FUNCTION_BLOCK FB_MatrixMultiplication
VAR_INPUT
	A : Matrix;
	B : Matrix;
END_VAR
VAR_OUTPUT
	out : Matrix;
END_VAR
VAR
	i : INT;
	j : INT;
	k : INT;
END_VAR

FOR i := 0 TO A.nRows-1 DO
    FOR j := 0 TO B.nCols-1 DO
        out.data[i, j] := 0; 
        FOR k := 0 TO B.nRows-1 DO
            out.data[i, j] := out.data[i, j] + A.data[i, k] * B.data[k, j]; 
        END_FOR
    END_FOR
END_FOR
out.nCols := B.nCols;
out.nRows := A.nRows;

END_FUNCTION_BLOCK

(* stored: Version 1.1.0.1, ProductVersion 3.1.4024.12
   POU FB_MatrixMultiplication: Id {14eaf4c8-522e-4b5f-ac55-8b0816371b8f}, SpecialFunc None *)
